{attribute 'qualified_only'}
{attribute 'strict'}
{attribute 'to_string'}
TYPE
StationName_e :
(
    Station100 := 1,
    Station110 := 2,
    Station120 := 3,
    Station130 := 4,
    Station140 := 5,
    Station150 := 6,
    Station160 := 7,
    Station170 := 8,
    Station180 := 9,
    Station190 := 10,
    Station200 := 11,
    Station210 := 12,
    Station220 := 13,
    Station230 := 14,
    Station240 := 15,
    Station250 := 16,
    Station260 := 17,
    Station270 := 18
);
END_TYPE

(* stored: Version 1.1.0.1, ProductVersion 3.1.4024.6
   EnumerationTextList StationName_e: Id {9c5c3967-f60b-4d52-bdf8-9d59f2175d7d} *)
